(* PLC project static_torsion.project, CODESYS CODESYS V3.5 SP17 Patch 3 *)
(* stored: creationDateTime 1970-01-01T00:00:00, modificationDateTime 2026-06-22T15:12:39.4699931 *)

{attribute 'qualified_only'}
VAR_GLOBAL  (* GVL *)
  DEBUG : BOOL := TRUE;
  ServoCommand : CTRL_ID;  (* Текущая команда управления сервоприводом *)
  State : S_STATE;  (* Слово состояния *)
  Control : S_CTRL;  (* Слово управления *)
  DQ_Control : PDQ_OLD;  (* Прямое управление дискретными выходами (используется только в сервисном режиме) *)
  UZ_Control : CTRL_ID;  (* Прямое управление сервоприводом (используется только в сервисном режиме) *)
  fbAlarm : ALARM;
  fbServo : SERVO;
  xLS_DOOR_EN : BOOL;  (* Если установлен, то контролировать открытие двери *)
  xLS_UP_EN : BOOL;  (* Если установлены, то контролировать КВ ВЕРХ и КВ НИЗ соответственно *)
  xLS_DN_EN : BOOL;  (* Если установлены, то контролировать КВ ВЕРХ и КВ НИЗ соответственно *)
  DI : PDI;  (* Входы дискретные модуль A11 (ECAT-2053) *)
  DQ : PDQ;  (* Выходы дискретные модуль A13 (ECAT-2057) *)
  iTorque_RAW : INT;  (* Значение момента с АЦП модуля *)
  rTorque : REAL;  (* Нескорректированное начение момента от тензодатдатчика в Нм. *)
  rTorqueCalibrated : REAL;  (* Скорректированное и масштабированное значение момента (модель и коэффициенты преобразования см. в функции расчета момента) *)
  iTorqueScaled : INT;  (* Скорректированное и масштабированное значение датчика момента (25000 = 50 Нм) *)
  udiEncoder_RAW : UDINT;  (* Угол: измеренное абсолютное значение в условных единицах датчика *)
  xPowerEnable : BOOL;  (* Управление приводом *)
  xMoveFollowExec : BOOL;
  xMoveRelativeExec : BOOL;
  xJogForwardExec : BOOL;
  xJogBackwardExec : BOOL;
  xResetExec : BOOL;
  xStopExec : BOOL;
  xHaltExec : BOOL;
  lrFollowVelocity : LREAL;
  lrRelativeVelocity : LREAL;
  lrRelativeDistance : LREAL;
  lrJogVelocity : LREAL;
  lrRelativeAcc : LREAL;
  lrRelativeDec : LREAL;
  lrJogAcc : LREAL;
  lrJogDec : LREAL;
  iTorqueSV : INT;
  iJogVelocity : INT;
  rActualTension : REAL;  (* Управление параметрами ПИД регулятора *)
  rSetValue : REAL;
  rYMin : REAL := -200;  (* %% *)
  rYMax : REAL := 200;  (* %% *)
  rY : REAL;
  iTorqueSensorRange : UINT := 50;  (* Диапазон датчика момента в Нм *)
  iTorque_ADC_offset : INT;  (* Смещение нулевого положения АЦП. Задается при вызове команды обнуления на этапе калибровки *)
  rA1 : REAL := 0;  (* Коэффициенты для модели аппроксимации датчика момента *)
  rB1 : REAL := 1;
  rC1 : REAL := 0;
  rA2 : REAL := 1;
  rB2 : REAL := 0;
  udiEncoderOffset : UDINT := 0;  (* Смещение нулевого положения датчика поворота *)
  KP : REAL := 10;  (* Коэффициенты ПИД регулятора *)
  KI : REAL := 0.1;
  KD : REAL := 0;
END_VAR
